// TIA Portal V18 export
ORGANIZATION_BLOCK "Startup"   // OB100, LAD, Startup
TITLE = "Complete Restart"
{ S7_Optimized_Access := 'TRUE' }
AUTHOR : HenriP
VERSION : 0.1
// stored: AutoNumber true, IsIECCheckEnabled false, SetENOAutomatically false
   VAR_INPUT
      LostRetentive : Bool;   // True if retentive data are lost
      LostRTC : Bool;   // True if date and time are lost
   END_VAR
   VAR_TEMP
      InitCall : Bool;
   END_VAR
BEGIN

REGION Network 1: Startup
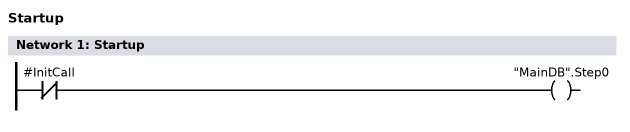
   RUNG wire#powerrail
      I_Contact( #InitCall )
      Coil( "MainDB".Step0 )
   END_RUNG
   // the same network as SCL:
   "MainDB".Step0 := NOT #InitCall;
END_REGION
END_ORGANIZATION_BLOCK
